Fanuc KAREL source: ko00044.KL

PROGRAM KO00044
%STACKSIZE=65535
%PRIORITY=65535
%NOLOCKGROUP
VAR
P1 : POSITION
P2 : XYZWPREXT
F : BOOLEAN
OUT : JOINTPOS9
BEGIN
F=TRUE
-- UNSAFE_SOURCE_IR line 11: CALL_RESULT MIRROR(convert_position_to_xyzwprext(P1), convert_xyzwprext_to_position(P2), F)
END KO00044
